// TIA Portal project "scl_7" (V18)

(* hardware
DEVICE "S7-1200 station_1"  S7-1200 Station
   slot 0: "Rack_0"  S7-1200 Rack  Rack  V1.0
   slot 1: "PLC_1"  CPU 1214C DC/DC/DC  6ES7 214-1AG40-0XB0  V4.6
*)

// ===== PLC "PLC_1"  CPU 1214C DC/DC/DC =====

VAR_GLOBAL   // PLC tag table "Default tag table"
   "kenar tetikleme merker" AT %M0.0 : Bool;
   "yardımcı kenar tetkileme merker" AT %M0.1 : Bool;
   "START" AT %I0.0 : Bool;
   "ÇIKIŞ" AT %Q0.0 : Bool;
   "STOP" AT %I0.1 : Bool;
END_VAR

FUNCTION "Block_1" : Void   // FC1, SCL
{ S7_Optimized_Access := 'TRUE' }
VERSION : 0.1
BEGIN
       "kenar tetikleme merker" := "START" AND NOT "yardımcı kenar tetkileme merker";

       "yardımcı kenar tetkileme merker" := "START";

       IF "kenar tetikleme merker" =1 THEN
           "ÇIKIŞ" := 1;
       ELSIF "STOP"=1 THEN
           "ÇIKIŞ" := 0;
       END_IF;
END_FUNCTION

ORGANIZATION_BLOCK "Main"   // OB1, LAD, ProgramCycle
TITLE = "Main Program Sweep (Cycle)"
{ S7_Optimized_Access := 'TRUE' }
VERSION : 0.1
// pozitif kenar tetikleme
   VAR_INPUT
      Initial_Call : Bool;   // Initial call of this OB
      Remanence : Bool;   // =True, if remanent data are available
   END_VAR
BEGIN

REGION Network 1
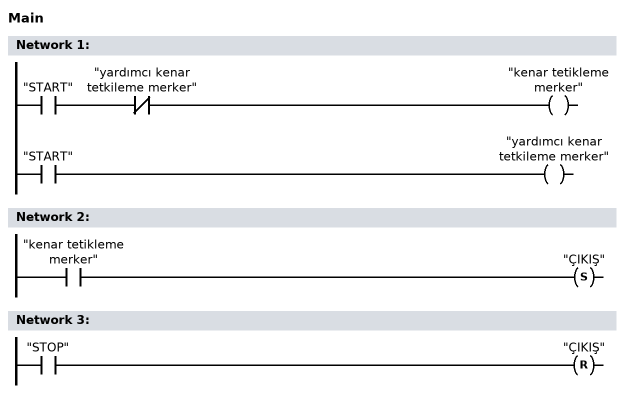
   RUNG wire#powerrail
      Contact( "START" )
      I_Contact( "yardımcı kenar tetkileme merker" )
      Coil( "kenar tetikleme merker" )
   END_RUNG
   RUNG wire#powerrail
      Contact( "START" )
      Coil( "yardımcı kenar tetkileme merker" )
   END_RUNG
   // the same network as SCL:
   "kenar tetikleme merker" := "START" AND NOT "yardımcı kenar tetkileme merker";
   "yardımcı kenar tetkileme merker" := "START";
END_REGION

REGION Network 2
   RUNG wire#powerrail
      Contact( "kenar tetikleme merker" )
      S_Coil( "ÇIKIŞ" )
   END_RUNG
   // the same network as SCL:
   IF "kenar tetikleme merker" THEN "ÇIKIŞ" := TRUE; END_IF;
END_REGION

REGION Network 3
   RUNG wire#powerrail
      Contact( "STOP" )
      R_Coil( "ÇIKIŞ" )
   END_RUNG
   // the same network as SCL:
   IF "STOP" THEN "ÇIKIŞ" := FALSE; END_IF;
END_REGION
END_ORGANIZATION_BLOCK